PROGRAM MBUS_WZaehler_Basement (* hier wird die Klemme, an welche der M-Bus mit den Zählern angeschlossen ist, alle 10ms aufgerufen *)
VAR
	Komm_Klemme_WZaehler_Basement 		: FB_MBUSKL6781;

	WMZ350								: FB_MBUS_General_Ext;
	WMZ305								: FB_MBUS_General_Ext;
	WMZ300								: FB_MBUS_General_Ext;
	WMZ100								: FB_MBUS_General_Ext;
	WMZ455								: FB_MBUS_General_Ext;
	WMZ245								: FB_MBUS_General_Ext;
	WMZ235								: FB_MBUS_General_Ext;
	WMZ425								: FB_MBUS_General_Ext;
		
	//basement
	adrWMZ350					: ST_MBus_SecAdr := (udiIdNumber:=16#75372672);
	adrWMZ305					: ST_MBus_SecAdr := (udiIdNumber:=16#75234689);
	adrWMZ100					: ST_MBus_SecAdr := (udiIdNumber:=16#75494412);
	adrWMZ300					: ST_MBus_SecAdr := (udiIdNumber:=16#75878308);
	
	adrWMZ455					: ST_MBus_SecAdr := (udiIdNumber:=16#75375855);
	adrWMZ245					: ST_MBus_SecAdr := (udiIdNumber:=16#75563317);
	adrWMZ235					: ST_MBus_SecAdr := (udiIdNumber:=16#13859503);
	adrWMZ425					: ST_MBus_SecAdr := (udiIdNumber:=16#75878305);
	
END_VAR

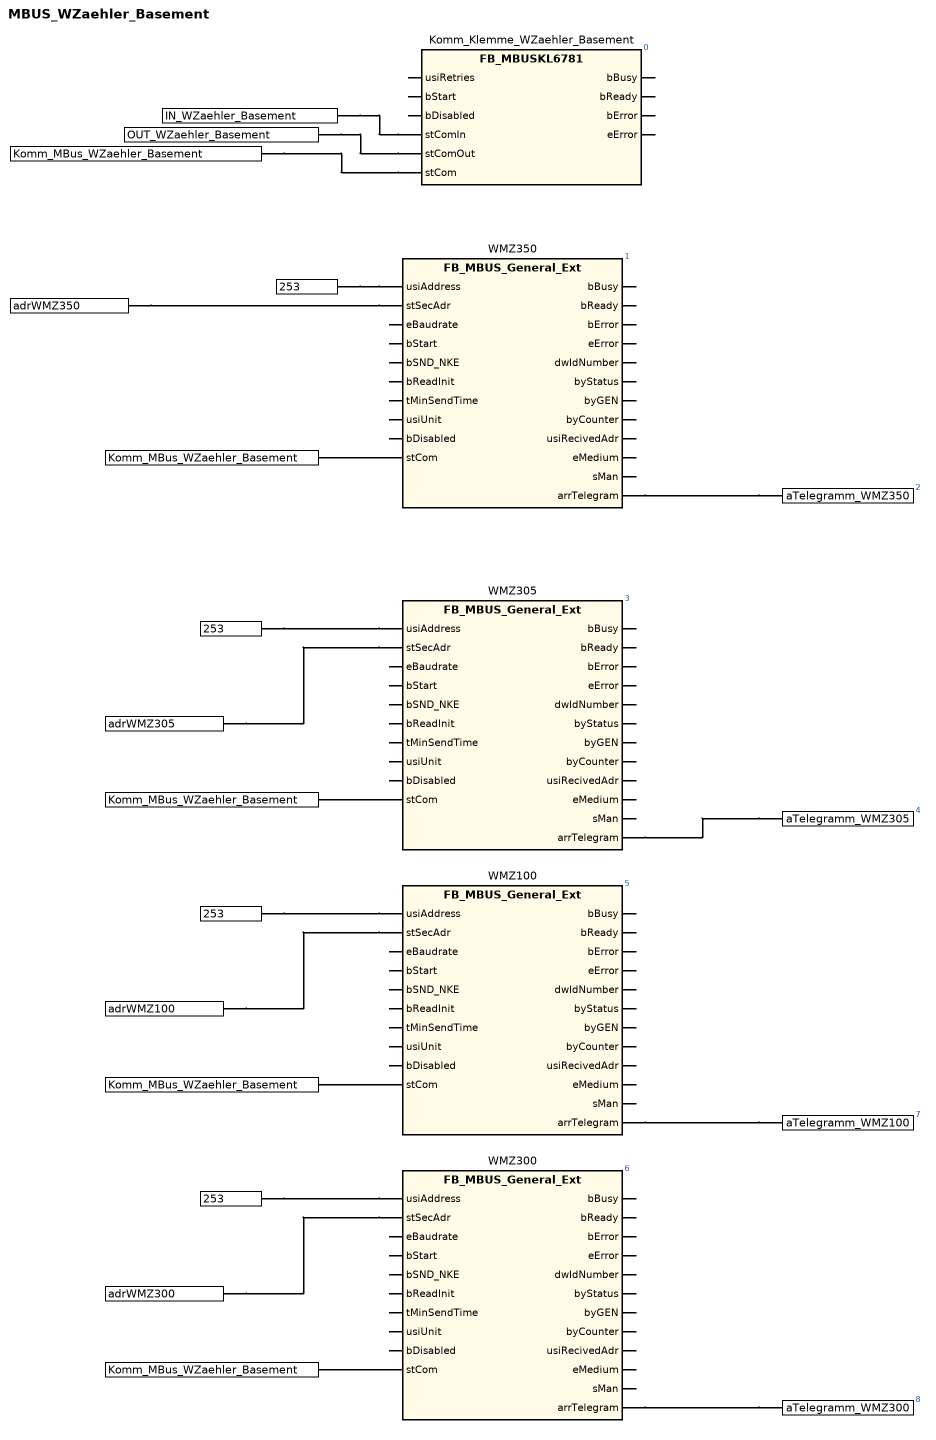
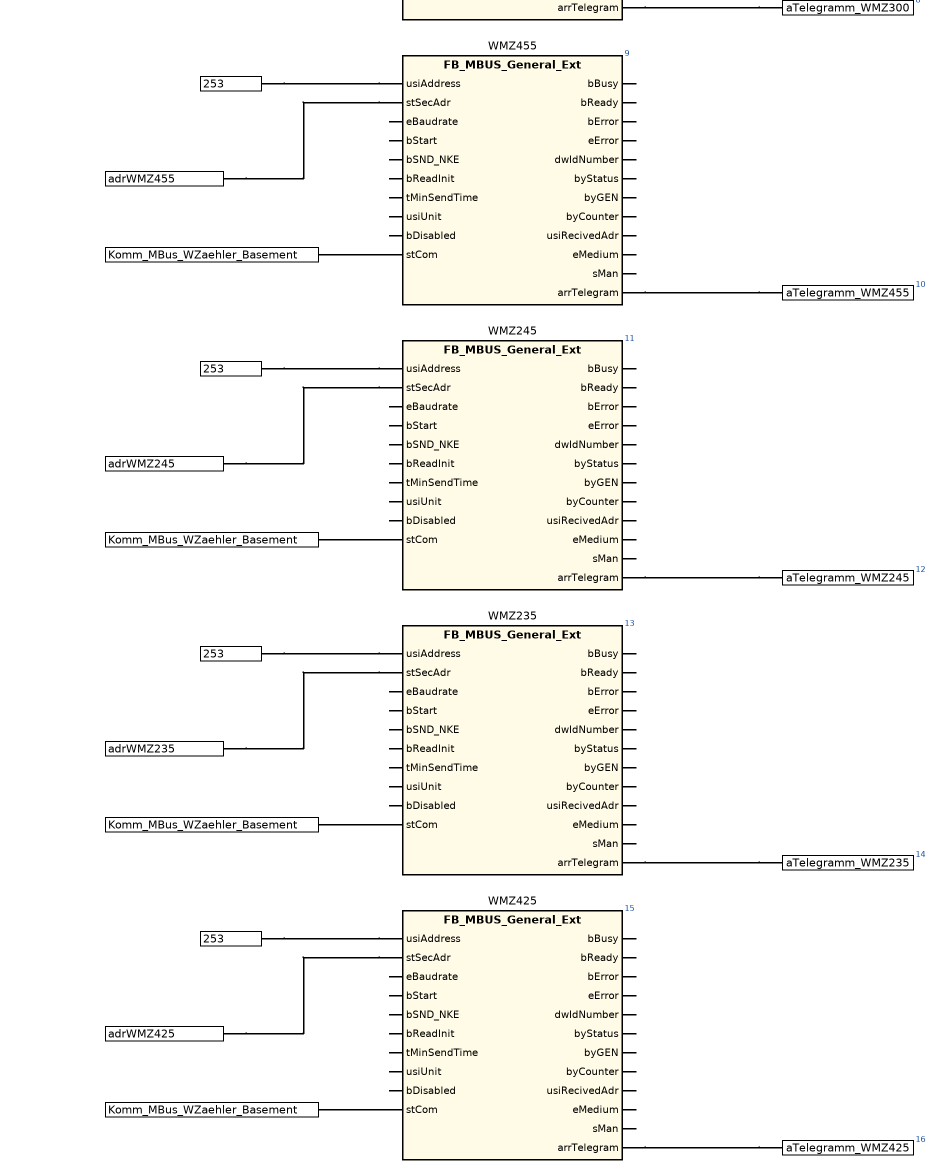
Komm_Klemme_WZaehler_Basement(
    stComIn := IN_WZaehler_Basement,
    stComOut := OUT_WZaehler_Basement,
    stCom := Komm_MBus_WZaehler_Basement); // FB_MBUSKL6781
WMZ350(usiAddress := 253, stSecAdr := adrWMZ350, stCom := Komm_MBus_WZaehler_Basement); // FB_MBUS_General_Ext
aTelegramm_WMZ350 := WMZ350.arrTelegram;
WMZ305(usiAddress := 253, stSecAdr := adrWMZ305, stCom := Komm_MBus_WZaehler_Basement); // FB_MBUS_General_Ext
aTelegramm_WMZ305 := WMZ305.arrTelegram;
WMZ100(usiAddress := 253, stSecAdr := adrWMZ100, stCom := Komm_MBus_WZaehler_Basement); // FB_MBUS_General_Ext
WMZ300(usiAddress := 253, stSecAdr := adrWMZ300, stCom := Komm_MBus_WZaehler_Basement); // FB_MBUS_General_Ext
aTelegramm_WMZ100 := WMZ100.arrTelegram;
aTelegramm_WMZ300 := WMZ300.arrTelegram;
WMZ455(usiAddress := 253, stSecAdr := adrWMZ455, stCom := Komm_MBus_WZaehler_Basement); // FB_MBUS_General_Ext
aTelegramm_WMZ455 := WMZ455.arrTelegram;
WMZ245(usiAddress := 253, stSecAdr := adrWMZ245, stCom := Komm_MBus_WZaehler_Basement); // FB_MBUS_General_Ext
aTelegramm_WMZ245 := WMZ245.arrTelegram;
WMZ235(usiAddress := 253, stSecAdr := adrWMZ235, stCom := Komm_MBus_WZaehler_Basement); // FB_MBUS_General_Ext
aTelegramm_WMZ235 := WMZ235.arrTelegram;
WMZ425(usiAddress := 253, stSecAdr := adrWMZ425, stCom := Komm_MBus_WZaehler_Basement); // FB_MBUS_General_Ext
aTelegramm_WMZ425 := WMZ425.arrTelegram;

END_PROGRAM

(* stored: Version 1.1.0.1, ProductVersion 3.1.4024.10
   POU MBUS_WZaehler_Basement: Id {3c9e8112-e798-4c93-b47a-0b8293d8b0d7}, SpecialFunc None *)
